PROGRAM MAIN
VAR
	fbIMU : FB_AccelerationSensor;
	
	x : REAL;
	y : REAL;
	z : REAL;
	
	acc : ARRAY [0..2] OF REAL;

//	fbEL6001	: FB_SerialCom;
	
//	(* exchange buffers with background communication with the PC COM port device *)
//	RxBufferPcCom	: ComBuffer;	(* Receive data buffer; used with all receive function blocks *)
//	TxBufferPcCom	: ComBuffer;	(* Transmit data buffer; used with all receive function blocks *)
	
//	acc_x : REAL;
//	acc_y : REAL;	
//	acc_z : REAL;
////	acc_x2 : REAL;
////	acc_y2 : REAL;	
////	acc_z2 : REAL;
////	acc_x3 : REAL;
////	acc_y3 : REAL;	
////	acc_z3 : REAL;
////	acc_x4 : REAL;
////	acc_y4 : REAL;	
////	acc_z4 : REAL;

//	fbTimer : TON;
//	fbReset : TON;
//	fbTrigger : R_TRIG;
//	iCounter1 : UDINT;
//	iCounter2 : UDINT;
//	a_iPackets : ARRAY [0..9] OF UDINT;
//	i : UDINT := 0;
//	iSum : UDINT := 0;
//	rPacketRate : REAL := 0;
//	bTrigger : BOOL := FALSE;
//	bCount : BOOL;

END_VAR

fbIMU();

acc := fbIMU.aAccelerationValues;

x := acc[0];
y := acc[1];
z := acc[2];



//fbEL6001(TxBuffer:=TxBufferEL, RxBuffer:=RxBufferEL);

//acc_x := fbEL6001.getAccelerationValueX;
//acc_y := fbEL6001.getAccelerationValueY;
//acc_z := fbEL6001.getAccelerationValueZ;

//acc_x2 := fbEL6001.getAccelerationValueX2;
//acc_y2 := fbEL6001.getAccelerationValueY2;
//acc_z2 := fbEL6001.getAccelerationValueZ2;

//acc_x3 := fbEL6001.getAccelerationValueX3;
//acc_y3 := fbEL6001.getAccelerationValueY3;
//acc_z3 := fbEL6001.getAccelerationValueZ3;

//acc_x4 := fbEL6001.getAccelerationValueX4;
//acc_y4 := fbEL6001.getAccelerationValueY4;
//acc_z4 := fbEL6001.getAccelerationValueZ4;

doPacketCount();					//start packet count by setting bCount 'true' --> rPacketRate shows average rate per second

METHOD doPacketCount : REAL
VAR_INPUT
END_VAR
//fbTimer(IN := bCount, PT := T#1S);
//fbTrigger(CLK := fbTimer.IN);

//IF fbTrigger.Q THEN
//	iCounter1 := fbEL6001.nReceiveCounter;
//END_IF

//IF fbTimer.Q THEN
//	iCounter2 := fbEL6001.nReceiveCounter;
//	a_iPackets[i] := iCounter2 - iCounter1;
//	iSum := iSum + a_iPackets[i];
//	i := i + 1;
//	bTrigger := TRUE;
//	bCount := FALSE;
//END_IF

//IF i = 10 THEN
//	bTrigger := FALSE;
//	rPacketRate := (UDINT_TO_REAL(iSum) / UDINT_TO_REAL(i));			//times amount of packets
//	i := 0;
//	iSum := 0;
//END_IF

//fbReset(IN := bTrigger, PT := T#3S);
//IF fbReset.Q THEN
//	bCount := TRUE;
//	bTrigger := FALSE;
//END_IF
END_METHOD

END_PROGRAM

(* stored: Version 1.1.0.1, ProductVersion 3.1.4024.12
   POU MAIN: Id {aef089b1-c7c5-479f-8336-a7bf9b8b2785}, SpecialFunc None
   Method doPacketCount: Id {f491d74c-1c83-4939-a57e-78d104db15c3} *)
